FUNCTION_BLOCK Test_AggregateResult_Starting EXTENDS T_UnitTestBase
VAR
    ResultAggregate : T_ResultAggregate;
    Execution1      : T_Execution;
    Execution2      : T_Execution;
    Execution3      : T_Execution;
END_VAR

METHOD Init
Execution1.FB_init(FALSE,FALSE);
Execution2.FB_init(FALSE,FALSE);
Execution3.FB_init(FALSE,FALSE);
END_METHOD

{attribute 'analysis' := '-33'} // inhibit unused variable warning
METHOD RunTest
VAR_OUTPUT
    TestCompleted : BOOL;
    TestFailed    : BOOL;
END_VAR
ResultAggregate.ClearResults();

ResultAggregate.AddResult(Execution1);
ResultAggregate.AddResult(Execution2);
ResultAggregate.AddResult(Execution3);

TestFailed S= NOT AssertFalse(Source    := TestName,
                              Condition := ResultAggregate.Starting,
                              Message   := 'ResultAggregate.Starting is not false',
                              Failed    =>);

Execution1.Start();

TestFailed S= NOT AssertTrue(Source    := TestName,
                             Condition := ResultAggregate.Starting,
                             Message   := 'ResultAggregate.Starting is false',
                             Failed    =>);

TestCompleted := TRUE;
END_METHOD

END_FUNCTION_BLOCK

(* stored: Version 1.1.0.1, ProductVersion 3.1.4024.12
   POU Test_AggregateResult_Starting: Id {37f7fd09-fcb5-44f2-86e4-0e4f8d59a3a3}, SpecialFunc None
   Method Init: Id {f37773dd-cb64-4e2d-9357-b2fae6f90d28}
   Method RunTest: Id {8d50d90d-e241-4c1e-a7be-6f7c1a112ae5} *)
